FUNCTION_BLOCK FB_CounterConsumer
VAR
    counter : B2SignedDelta_Plc.FB_Counter;
    delta : DINT;
END_VAR

delta := UDINT_TO_DINT(counter.GetSignedDelta(a := 5, b := 7));

END_FUNCTION_BLOCK

(* stored: Version 1.1.0.1
   POU FB_CounterConsumer: Id {f561e0c3-f2ca-4cff-902d-8728c72c678d}, SpecialFunc None *)
